// Mitsubishi GX Works2 project: mov_dmov   PLC: Q03UDV

PROGRAM MAIN
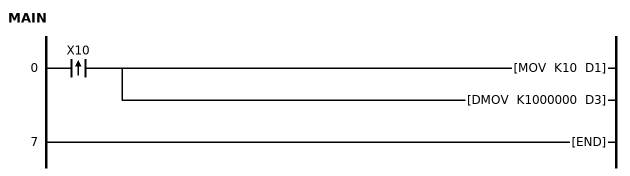
0     LDP     X10
      MOV     K10 D1
      DMOV    K1000000 D3
7     END
END_PROGRAM
